Fanuc KAREL source: kb00178.KL

-- PROVISIONAL review KL for V770-1; original PC SHA256 58afa8855a5f9ed0a504cd0c64d040c24e9297b9c2439aeaeb3d421061cf96e9
-- Incomplete behavior may be omitted. Consult companion uncertainty JSON. Do not deploy.
PROGRAM KB00178
%NOLOCKGROUP
BEGIN
  -- UNRESOLVED_PC offsets 5-12; opcodes 9D,23
  -- UNRESOLVED_PC offsets 17-28; opcodes 2E,23
  -- UNRESOLVED_PC offsets 33-40; opcodes 9D,23
  -- UNRESOLVED_PC offsets 45-67; opcodes 27,22,22,22,31
  -- UNRESOLVED_PC offsets 72-76; opcodes 7F
END KB00178
